FUNCTION_BLOCK FB_PID
VAR_INPUT
	fX : LREAL;
	fXReal : LREAL;
	fSignalIntegrated : LREAL;
	fSignalDerivated : LREAL;
	fKp : LREAL;
	fKi : LREAL;
	fKd : LREAL;
END_VAR
VAR_OUTPUT
	fSignalI : LREAL;
	fSignalD : LREAL;
	fSignalAdjusted : LREAL;
	fError  : LREAL;
END_VAR
VAR
	fTempP : LREAL;
	fTempI : LREAL;
	fTempD : LREAL;
	fTempOut : LREAL;
END_VAR

fError := fX - fXReal;

fSignalI := fError;
fSignalD := fError;

fTempP := fError * fKp;
fTempI := fSignalIntegrated * fKi;
fTempD := fSignalDerivated * fKd;

fTempOut := fTempP + fTempI + fTempD;

IF fTempOut > 1.0 THEN
	fSignalAdjusted := 1.0;
ELSIF fTempOut < -1.0 THEN
	fSignalAdjusted := -1.0;
ELSE
	fSignalAdjusted := fTempOut;
END_IF

END_FUNCTION_BLOCK

(* stored: Version 1.1.0.1, ProductVersion 3.1.4024.13
   POU FB_PID: Id {c3b9a6ed-2e03-46aa-9312-a6c1264b90f3}, SpecialFunc None *)
